PROGRAM PRG_PanelDeControl
VAR
	tRTrigSacar			: R_TRIG;

	i: INT := 1;
	bReset : BOOL;
	iSolicitudColor: COLOR;
END_VAR

VAR_INPUT
	iSolicitud: INT := 0;
END_VAR

tRTrigSacar(CLK:= GVL_Almacen.Sacar);

(* Aquí sumamos el número de cajas a sacar, que nunca puede ser mayor de las que hay *)

IF tRTrigSacar.Q THEN
	iSolicitud := iSolicitud + 1;
END_IF

(* BOTÓN NARANJA. Paro fin de ciclo *)

IF GVL_Almacen.bReset THEN
	bReset := TRUE;
END_IF

IF bReset AND PRG_RetiradaAlmacen.SELECCION > 2 THEN
		iSolicitud := 1;
END_IF


(* Rosca de selección del tipo de caja *)
	
IF GVL_Almacen.sSelector.StateAzul THEN
	GVL_Almacen.LedAzul := TRUE;
	GVL_Almacen.LedVerde := FALSE;
	GVL_Almacen.LedMetal := FALSE;
	iSolicitudColor := AZUL;
	GVL_Almacen.iDisplay := PRG_Almacen.iCantidadAzul;
END_IF

IF NOT GVL_Almacen.sSelector.StateMetal AND NOT GVL_Almacen.sSelector.StateAzul THEN
	GVL_Almacen.LedAzul := FALSE;
	GVL_Almacen.LedVerde := TRUE;
	GVL_Almacen.LedMetal := FALSE;
	iSolicitudColor := VERDE;
	GVL_Almacen.iDisplay := PRG_Almacen.iCantidadVerde;
END_IF

IF GVL_Almacen.sSelector.StateMetal THEN
	GVL_Almacen.LedAzul := FALSE;
	GVL_Almacen.LedVerde := FALSE;
	GVL_Almacen.LedMetal := TRUE;
	iSolicitudColor := METAL;
	GVL_Almacen.iDisplay := PRG_Almacen.iCantidadMetal;
END_IF

END_PROGRAM

(* stored: Version 1.1.0.1, ProductVersion 3.1.4024.12
   POU PRG_PanelDeControl: Id {4125b4fd-54c0-4476-b867-203b20e49183}, SpecialFunc None *)
